(* PLC project v0.6.04_CycleSemiAuto.project, CODESYS CODESYS V3.5 SP19 Patch 1 *)
(* stored: creationDateTime 2026-07-24T00:33:51.925669, modificationDateTime 2026-07-24T00:33:51.925669 *)

(* ═══════════════════════════════════════════════════════════════ 🔧 ST_WinchCfg — Configurations et paramètres réglables pour un Treuil M1/M2 ─────────────────────────────────────────────────────────────── 🎨 Destiné au paramétrage et calibration depuis l'IHM (RETAIN). 📄 2026-07-24 : CfgMaxStepDescente/CfgMaxStepAscent/CfgSlowdownDistance_M/CfgSlowSpeed_Pct déplacés vers GVL_IHM.Commun.Cfg (WinchMaxStepDescente/etc.) — étaient partagés M1/M2 via réconciliation ad-hoc, une seule instance dans Commun élimine le besoin de réconciliation. ═══════════════════════════════════════════════════════════════ *)
TYPE ST_WinchCfg : STRUCT
  CfgTopSensorPos_M : REAL := 8.5;  (* 📐 Position cible du capteur haut (m) *)
  CfgHomingTarget_M : REAL := 0;  (* 🔧 Cible libre Homing unitaire MAINT_N2 [-99..+99 m] *)
  CfgRampAccelRate : REAL := 50;  (* 📈 Rampe d'accélération (%/s) *)
  CfgRampDecelNormalRate : REAL := 150;  (* 📉 Rampe de décélération normale (%/s) *)
  CfgRampDecelFastRate : REAL := 400;  (* ⚡ Rampe de décélération rapide / SafeStop (%/s) *)
  CfgCableLimitDescent_M : REAL := -20;  (* 📐 Limite basse physique de descente (m, négatif) *)
  CfgCableLimitAscent_M : REAL := 6.75;  (* 📐 Limite haute d'exploitation NORMALE (m) -- REX 2026-08-07 (25), aligné sur GVL_PERSISTENT *)
  Initialized : BOOL := FALSE;  (* 🐛 FIX 2026-07-23 : flag restauration boot (défaut FALSE non ambigu, contrairement à un champ métier dont le défaut peut valoir n'importe quoi) — PRG_SUPERVISION_CFC.st §2/§3 🚦 TRUE = config restaurée depuis GVL_PERSISTENT ce boot *)
END_STRUCT;
END_TYPE

(* ═══════════════════════════════════════════════════════════════ 🌉 FB_CfgPersistBridge_WinchCfg — Pont persistance générique pour ST_WinchCfg ─────────────────────────────────────────────────────────────── 🎯 Deux instances indépendantes : M1TreuilRetenue.Cfg et M2TreuilBenne.Cfg. Restaure Persist → Hmi au boot si nécessaire, puis sauvegarde Hmi → Persist. ═══════════════════════════════════════════════════════════════ *)
FUNCTION_BLOCK FB_CfgPersistBridge_WinchCfg
  VAR_OUTPUT
    JustRestored : BOOL;  (* 🔔 TRUE pendant le scan de restauration *)
  END_VAR
  VAR_IN_OUT
    Hmi : ST_WinchCfg;  (* 🖥️ Struct exposé à l'IHM *)
    Persist : ST_WinchCfg;  (* 💾 Mémoire PERSISTENT *)
  END_VAR

            

JustRestored := FALSE;
IF NOT Hmi.Initialized THEN
    Hmi := Persist;
    Hmi.Initialized := TRUE;
    JustRestored := TRUE;
ELSE
    Persist := Hmi;
END_IF;

          
END_FUNCTION_BLOCK
